FUNCTION_BLOCK PUBLIC FB_AUT_ABSTRACT IMPLEMENTS IProcessSampleMover
    (****************************************************************************)
    (*	POU_AUT_zxx			Bausteinaufrufe Station	zxx							*)
    (*	Status				ungetestet											*)
    (*  Version:			1.0													*)
    (*	Beschrieb:																*)
    (*																			*)
    (*	Abläufe:			FB_ABLzxxA		Hauptablauf							*)
    (*																			*)
    (*																			*)
    (* 	25.09.2019/Dj															*)
    (****************************************************************************)
    (*	dd.mm.yyyy   KZ    x.y			Beschrieb								*)
    (****************************************************************************)
VAR_INPUT
    (* standart Eingänge *)
    xIN_Init       : BOOL;    // Initialisieren	
    xIN_Quit       : BOOL;    // Fehler quittieren 
    xIN_Start      : BOOL;    // Schrittkette Starten
    xIN_Step       : BOOL;    // Schrittkette Starten/Nachster Schritt
    xIN_ManuCycle  : BOOL;    // Zylus Manuell Starten
    xIN_AlarmAktiv : BOOL;    // Alarm aktiv 
    xIN_DryCycle   : BOOL;    // Fahren ohne Teile 
    enIN_State     : enState; // Status Anlage/Zelle 
    tIN_Timeout    : TIME;    // Timout 
    xIN_On         : BOOL;    // Station eingeschaltet 

    (* spezifische Eingänge *)

END_VAR
VAR_OUTPUT
    (* standart Ausgänge *)
    xOUT_InitDone : BOOL; // fertig initialisiert
    xOUT_Done     : BOOL; // alle Abläufe fertig
    xOUT_Ready    : BOOL; // Station ist bereit (wartet auf Start)
    xOUT_ErrFlag  : BOOL; // Error Flag   
    xOUT_Wait     : BOOL; // alle Abläufe warten
    xOUT_AlarmST  : BOOL; // Station hat Alarm

    (* spezifische Ausgänge *)

END_VAR
VAR

    (* Flags *)
    xReset     : BOOL; // Schrittketten zurücksetzen
    xManuCycle : BOOL; // Manueller Zylus aktiv	
    xNextStep  : BOOL; // Nächster Schritt erlaubt	

    xDummy : BOOL := TRUE; // Platzhalter		

    i : INT;

    _iID : INT := 0; // instance ID, is set during FB_Init using the value of _iInstanceCounter 

    _ProcessExecution : ProcessExecution_e := ProcessExecution_e.ExecuteImmediately;

    _Mover            : REFERENCE TO FB_Mover;
    _xMoverShouldLeave : BOOL; // flag to synchronise process and MoverMan, MoverMan needs to call TakeMover() to reset this flag

END_VAR
VAR_STAT
    _iInstanceCounter : INT := 1; // instance counter
END_VAR

METHOD Equals : BOOL
VAR_INPUT
    object : ANY;
END_VAR
Equals := THIS = object.pValue;
END_METHOD

METHOD FB_init : BOOL
VAR_INPUT
	bInitRetains : BOOL; // if TRUE, the retain variables are initialized (warm start / cold start)
	bInCopyCode : BOOL;  // if TRUE, the instance afterwards gets moved into the copy code (online change)
END_VAR
THIS^._iID := THIS^._iInstanceCounter;
THIS^._iInstanceCounter := THIS^._iInstanceCounter +1;
END_METHOD

METHOD GiveMover : IProcessSampleMover
VAR_INPUT
	mover : REFERENCE TO FB_Mover;
END_VAR
THIS^._Mover REF= mover;
END_METHOD

(* % of completion of the process *)
PROPERTY iCompletionPC : INT
GET
END_GET
END_PROPERTY

(* Process time, expressed in milisecond *)
PROPERTY iProcessTimeMili_1 : DINT
GET
END_GET
SET
END_SET
END_PROPERTY

(* Process time, expressed in milisecond *)
PROPERTY iProcessTimeMili_2 : DINT
GET
END_GET
SET
END_SET
END_PROPERTY

PROPERTY Mover : REFERENCE TO FB_Mover
GET
Mover REF= THIS^._Mover;
END_GET
SET
THIS^._Mover REF= Mover;
END_SET
END_PROPERTY

PROPERTY PUBLIC ProcessExecution : ProcessExecution_e
GET
ProcessExecution := THIS^._ProcessExecution;
END_GET
SET
THIS^._ProcessExecution := ProcessExecution;
END_SET
END_PROPERTY

METHOD TakeMover : IProcessSampleMover
THIS^.Mover REF= 0;
THIS^._xMoverShouldLeave := FALSE;
END_METHOD

METHOD ToString : STRING
VAR_INPUT
END_VAR
VAR
END_VAR
ToString := CONCAT('FB_AUT_ABSTRACT_', TO_STRING(THIS^._iID));
END_METHOD

PROPERTY xBusy : BOOL
GET
END_GET
SET
END_SET
END_PROPERTY

PROPERTY xDone : BOOL
GET
END_GET
END_PROPERTY

PROPERTY xMoverPathFree : BOOL
GET
END_GET
END_PROPERTY

PROPERTY xMoverShouldLeave : BOOL
GET
END_GET
END_PROPERTY

END_FUNCTION_BLOCK

(* stored: Version 1.1.0.1, ProductVersion 3.1.4024.12
   POU FB_AUT_ABSTRACT: Id {e9f820e2-63e4-4738-93a0-905f1e9dea0a}, SpecialFunc None
   Method Equals: Id {8bac0c73-0ccf-4b73-b532-5308ec23070b}
   Method FB_init: Id {657b0df4-0f9d-41d9-87f9-0136e5aa09ba}
   Method GiveMover: Id {d729fa09-00f6-4fc7-85c9-8b734ecb221f}
   Property iCompletionPC: Id {8e22b084-7383-488c-96f6-894a84f0ff6f}
   Get Get: Id {ed468f8e-ad8e-4266-9111-dfce9ece96d5}
   Property iProcessTimeMili_1: Id {00789763-b0c1-46da-b435-85ea24c17c60}
   Get Get: Id {804867bb-2eb1-42d5-be2d-daa9d1665638}
   Set Set: Id {1517f5af-3a45-47e8-823c-2d24b76bb472}
   Property iProcessTimeMili_2: Id {8a91a320-6ef0-40f0-9503-6d27209218cd}
   Get Get: Id {0978e08d-b31b-4f3e-a166-9c86b7369801}
   Set Set: Id {024d548c-93a8-478e-9a9a-92f21b77cdbd}
   Property Mover: Id {9d530e94-74ee-4547-a5fe-415f2b499bca}
   Get Get: Id {bb9a0d39-fe92-4058-97d5-e050b0496d3c}
   Set Set: Id {b8fd65c4-0c02-4668-889e-b821e1ce887b}
   Property ProcessExecution: Id {bb49a628-8a3f-4bab-9d47-e6d291975a1b}
   Get Get: Id {c448a1fd-c6c8-4395-9e08-aa6ef2c00017}
   Set Set: Id {b70a4e0c-8b62-44e1-bd66-21e6ab166232}
   Method TakeMover: Id {4b449397-8235-4f7b-974a-5033a1ab7c6b}
   Method ToString: Id {b8f24df3-0394-4666-b4ef-41086ff75475}
   Property xBusy: Id {74f36b79-cf92-4973-a1ae-9b817a07ead9}
   Get Get: Id {350150f3-ec85-49f2-ab2a-3ce0f560f39f}
   Set Set: Id {899959ff-8518-42e2-b770-7cb264186129}
   Property xDone: Id {aa707ad9-32ef-4678-ac04-381eab7d05fd}
   Get Get: Id {91d48dbe-c7e8-4220-a0fd-66cc33ecf52a}
   Property xMoverPathFree: Id {186cf167-6687-4650-8500-ed37470b16c8}
   Get Get: Id {93d97871-25b7-4a3b-9750-6db7069a86e9}
   Property xMoverShouldLeave: Id {dd9d11c3-6b68-4291-b1db-308c5d0878a1}
   Get Get: Id {4fd8e361-b39f-486c-8b35-94d9850bb1bf} *)
